(* IEC 61131-3 sources: Elmo_Master/Lasal_PRG/MotionTCPDemo/Class/Merker, 1 file *)

(* ---- Merker.st ---- *)
(*!
<Class
	Name               = "Merker"
	Revision           = "1.0"
	RealtimeTask       = "false"
	CyclicTask         = "false"
	BackgroundTask     = "false"
	Sigmatek           = "true"
	OSInterface        = "false"
	HighPriority       = "false"
	Automatic          = "false"
	UpdateMode         = "Prescan"
	IconPath           = ".\Class\Merker\Merker.ICO"
	SharedCommandTable = "true"
	Objectsize         = "(284,120)"
	Comment            = "to store data, not constant, not retentive">
	<Channels>
		<Server Name="Data" Visualized="true" Initialize="true" WriteProtected="false" Retentive="false"/>
	</Channels>
	<Dependencies>
		<Files>
			<File Path=".\Class\Ram\Ram.h" Include="false"/>
		</Files>
	</Dependencies>
</Class>
*)
Merker : CLASS
  //Servers:
	Data 	: SvrChCmd_DINT;
  //Clients:
  //Variables:
  //Functions:
  //Tables:
	FUNCTION @STD
		VAR_OUTPUT
			ret_code	: CONFSTATES;
		END_VAR;
	FUNCTION GLOBAL TAB @CT_;
END_CLASS;
